// TIA Portal V20 export
FUNCTION_BLOCK "Sequence_4_STKInterface"   // FB181, LAD
TITLE = Sequence
// Sequence template programmend in ladder logic
// stored: IsIECCheckEnabled true, MemoryReserve 100, Namespace Unit1.Em7, SetENOAutomatically true
   VAR_OUTPUT
      safeState : Bool;
   END_VAR
   VAR_IN_OUT
      controlNodeStep : "LER_typeStep";
      controlNodeJobs : "LAF_typeJobs";
      controlNodeSequence : "LAF_typeSequence";
      HmiInterfaceJobs : "LAF_typeJobsInterface";
      HmiInterfaceSequence : "LAF_typeSequenceInterface";
      PartDataStkPpPos : "LER_typePartData";
      InterfaceR2SData : "LER_typeCommunicationR2SData";
      InterfaceS2RData : "LER_typeCommunicationS2RData";
   END_VAR
   VAR
      instSequenceLADControl { ExternalWritable := 'False'} : "LAF_ControlLadSequence";
      instSequenceLADStatus { ExternalWritable := 'False'} : "LAF_StatusLadSequence";
      statPulse { ExternalWritable := 'False'} : Array[0..999] of Bool;
      statTonTimer { ExternalWritable := 'False'} : Array[0..999] of TON_TIME;
   END_VAR
   VAR_TEMP
      tempCustomerAction : Bool;   // Placeholder for possible actions
      tempDo_nothing_and_wait_for_init : Bool;   // Placeholder for doing nothing
      tempSafeStateCondition : Bool;   // Temp Condition for the equipment module to be in a safe state
      tempPartDataStkPpPos : "LER_typePartData";
   END_VAR
   VAR CONSTANT
      STEP_IDLE : DInt := 1;   // Idle Step
      JOB_1_STEP_01 : DInt := 101;
      JOB_1_STEP_11 : DInt := 111;
      JOB_1_STEP_21 : DInt := 121;
      JOB_1_STEP_31 : DInt := 131;
      JOB_1_STEP_41 : DInt := 141;
      JOB_1_STEP_51 : DInt := 151;
      JOB_1_STEP_61 : DInt := 161;
      JOB_1_STEP_71 : DInt := 171;
      JOB_1_STEP_81 : DInt := 181;
      JOB_1_STEP_91 : DInt := 191;
      JOB_2_STEP_01 : DInt := 201;
      JOB_2_STEP_11 : DInt := 211;
      JOB_2_STEP_21 : DInt := 221;
      JOB_2_STEP_31 : DInt := 231;
      JOB_2_STEP_41 : DInt := 241;
      JOB_2_STEP_51 : DInt := 251;
      JOB_2_STEP_61 : DInt := 261;
      JOB_2_STEP_71 : DInt := 271;
      JOB_2_STEP_81 : DInt := 281;
      JOB_2_STEP_91 : DInt := 291;
      JOB_3_STEP_01 : DInt := 301;
      JOB_3_STEP_11 : DInt := 311;
      JOB_3_STEP_21 : DInt := 321;
      JOB_3_STEP_31 : DInt := 331;
      JOB_3_STEP_41 : DInt := 341;
      JOB_3_STEP_51 : DInt := 351;
      JOB_3_STEP_61 : DInt := 361;
      JOB_3_STEP_71 : DInt := 371;
      JOB_3_STEP_81 : DInt := 381;
      JOB_3_STEP_91 : DInt := 391;
      JOB_4_STEP_01 : DInt := 401;
      JOB_4_STEP_11 : DInt := 411;
      JOB_4_STEP_21 : DInt := 421;
      JOB_4_STEP_31 : DInt := 431;
      JOB_4_STEP_41 : DInt := 441;
      JOB_4_STEP_51 : DInt := 451;
      JOB_4_STEP_61 : DInt := 461;
      JOB_4_STEP_71 : DInt := 471;
      JOB_4_STEP_81 : DInt := 481;
      JOB_4_STEP_91 : DInt := 491;
      STEP_IMMEDIATE_STOP : DInt := 901;   // Step executed when an immediate stop command is triggered for the sequence (i.e. when unit is in state aborting)
      SeqDelayTime : Time := T#100ms;
      SeqNoDelayTime : Time;
      TRUE : Bool := TRUE;
      FALSE : Bool := FALSE;
   END_VAR
   // // InterfaceR2SData.InterfaceData."Bool"[0] : Load Enable
   // // InterfaceR2SData.InterfaceData."Bool"[1] : Load Complete Comfirm
   // // InterfaceR2SData.InterfaceData."Bool"[2] : Cell Data Report
   // // InterfaceR2SData.InterfaceData."Bool"[10] : CollisionAreaOn
   // // InterfaceR2SData.InterfaceData."Bool"[11] : CollisionAreaOff
   // // InterfaceR2SData.InterfaceData."Bool"[15] : HeartBeat
   // // InterfaceS2RData.InterfaceData."Bool"[0] : Load Requset
   // // InterfaceS2RData.InterfaceData."Bool"[1] : Load Busy
   // // InterfaceS2RData.InterfaceData."Bool"[2] : Load Complete
   // // InterfaceS2RData.InterfaceData."Bool"[3] : Cell Data Request
   // // InterfaceS2RData.InterfaceData."Bool"[4] : Cell Data Report Ack
   // // InterfaceS2RData.InterfaceData."Bool"[5] : Cell Data Report Nck
   VAR_TEMP   // added for the SCL form of the ladder/FBD networks
      _w1 : Bool;
      _w2 : Bool;
      _w3 : Bool;
   END_VAR
BEGIN

REGION Network 1: BLOCK INFO HEADER
   // (company) / (C) Copyright (year)
   // ---------------------------------------------------------------------------------
   // Title:                             (Title of this block)
   // Comment/Function: (that is implemented in the block)
   // Library/Family:           (that the source is dedicated to)
   // Author:                        (department / person in charge / contact)
   // Target System:          (test system with FW version)
   // Engineering:              TIA Portal (SW version)
   // Restrictions:               (OB types, etc.)
   // Requirements:           (hardware, technological package, etc.)
   // ---------------------------------------------------------------------------------
   // Change log table:
   // Version          | Date             | Signature      | Expert in charge  | Changes applied ------------------------|----------------------|-------------------------|--------------------------------|-----------------------
   // 001.000.000 | yyyy-mm-dd | 0x00000000 | (name of expert) | First released version
END_REGION

REGION Network 2: DESCRIPTION
   // This is a template block provided by the Automation Framework. It can be used to create an own project.
   // The Block Info Header is prepared to put in your own data.
   // Description of the block could be added here and the docu created by Code2Docu.
END_REGION

REGION Network 3: *************** CONTROL **********************
END_REGION

REGION Network 4: Sequence Control
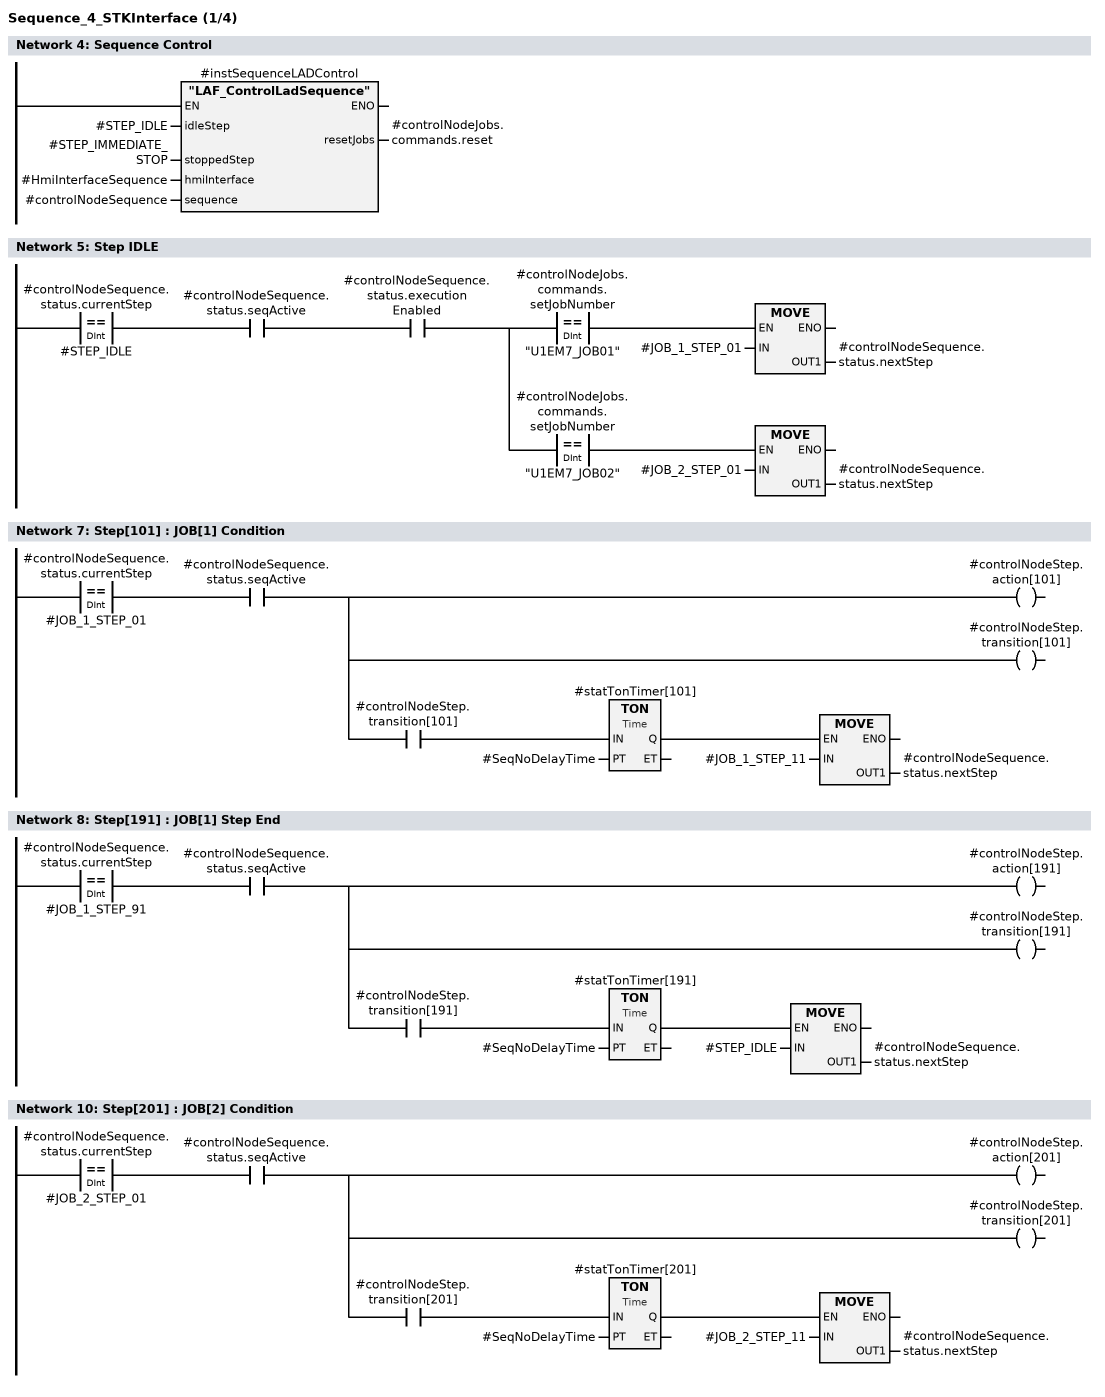
   RUNG wire#powerrail
      #instSequenceLADControl(idleStep := #STEP_IDLE, stoppedStep := #STEP_IMMEDIATE_STOP, hmiInterface := #HmiInterfaceSequence, sequence := #controlNodeSequence, resetJobs => #controlNodeJobs.commands.reset)
   END_RUNG
   // the same network as SCL:
   #instSequenceLADControl(idleStep := #STEP_IDLE,   // "LAF_ControlLadSequence"
                           stoppedStep := #STEP_IMMEDIATE_STOP,
                           hmiInterface := #HmiInterfaceSequence,
                           sequence := #controlNodeSequence,
                           resetJobs => #controlNodeJobs.commands.reset);
END_REGION

REGION Network 5: Step IDLE
   RUNG wire#powerrail
      { S7_Templates := "SrcType := DInt" } EQ_Contact(in1 := #controlNodeSequence.status.currentStep, in2 := #STEP_IDLE)
      Contact( #controlNodeSequence.status.seqActive )
      Contact( #controlNodeSequence.status.executionEnabled )
      wire#w1
      { S7_Templates := "SrcType := DInt" } EQ_Contact(in1 := #controlNodeJobs.commands.setJobNumber, in2 := "U1EM7_JOB01")
      Move(in := #JOB_1_STEP_01, out1 => #controlNodeSequence.status.nextStep)
   END_RUNG
   RUNG wire#w1
      { S7_Templates := "SrcType := DInt" } EQ_Contact(in1 := #controlNodeJobs.commands.setJobNumber, in2 := "U1EM7_JOB02")
      Move(in := #JOB_2_STEP_01, out1 => #controlNodeSequence.status.nextStep)
   END_RUNG
   // the same network as SCL:
   #_w1 := (#controlNodeSequence.status.currentStep = #STEP_IDLE) AND #controlNodeSequence.status.seqActive AND #controlNodeSequence.status.executionEnabled;
   IF #_w1 AND (#controlNodeJobs.commands.setJobNumber = "U1EM7_JOB01") THEN
       #controlNodeSequence.status.nextStep := #JOB_1_STEP_01;
   END_IF;
   IF #_w1 AND (#controlNodeJobs.commands.setJobNumber = "U1EM7_JOB02") THEN
       #controlNodeSequence.status.nextStep := #JOB_2_STEP_01;
   END_IF;
END_REGION

REGION Network 6: ******************** JOB[1] EM INITIALIZED ********************
END_REGION

REGION Network 7: Step[101] : JOB[1] Condition
   RUNG wire#powerrail
      { S7_Templates := "SrcType := DInt" } EQ_Contact(in1 := #controlNodeSequence.status.currentStep, in2 := #JOB_1_STEP_01)
      Contact( #controlNodeSequence.status.seqActive )
      wire#w1
      Coil( #controlNodeStep.action[101] )
   END_RUNG
   RUNG wire#w1
      Coil( #controlNodeStep.transition[101] )
   END_RUNG
   RUNG wire#w1
      Contact( #controlNodeStep.transition[101] )
      { S7_Templates := "time_type := Time" } #statTonTimer[101].TON(pt := #SeqNoDelayTime, et =>)
      Move(in := #JOB_1_STEP_11, out1 => #controlNodeSequence.status.nextStep)
   END_RUNG
   // the same network as SCL:
   #controlNodeStep.action[101] := (#controlNodeSequence.status.currentStep = #JOB_1_STEP_01) AND #controlNodeSequence.status.seqActive;
   #controlNodeStep.transition[101] := (#controlNodeSequence.status.currentStep = #JOB_1_STEP_01) AND #controlNodeSequence.status.seqActive;
   #statTonTimer[101].TON(IN := (#controlNodeSequence.status.currentStep = #JOB_1_STEP_01) AND #controlNodeSequence.status.seqActive AND #controlNodeStep.transition[101],
                          PT := #SeqNoDelayTime);
   IF #statTonTimer[101].Q THEN #controlNodeSequence.status.nextStep := #JOB_1_STEP_11; END_IF;
END_REGION

REGION Network 8: Step[191] : JOB[1] Step End
   RUNG wire#powerrail
      { S7_Templates := "SrcType := DInt" } EQ_Contact(in1 := #controlNodeSequence.status.currentStep, in2 := #JOB_1_STEP_91)
      Contact( #controlNodeSequence.status.seqActive )
      wire#w1
      Coil( #controlNodeStep.action[191] )
   END_RUNG
   RUNG wire#w1
      Coil( #controlNodeStep.transition[191] )
   END_RUNG
   RUNG wire#w1
      Contact( #controlNodeStep.transition[191] )
      { S7_Templates := "time_type := Time" } #statTonTimer[191].TON(pt := #SeqNoDelayTime, et =>)
      Move(in := #STEP_IDLE, out1 => #controlNodeSequence.status.nextStep)
   END_RUNG
   // the same network as SCL:
   #controlNodeStep.action[191] := (#controlNodeSequence.status.currentStep = #JOB_1_STEP_91) AND #controlNodeSequence.status.seqActive;
   #controlNodeStep.transition[191] := (#controlNodeSequence.status.currentStep = #JOB_1_STEP_91) AND #controlNodeSequence.status.seqActive;
   #statTonTimer[191].TON(IN := (#controlNodeSequence.status.currentStep = #JOB_1_STEP_91) AND #controlNodeSequence.status.seqActive AND #controlNodeStep.transition[191],
                          PT := #SeqNoDelayTime);
   IF #statTonTimer[191].Q THEN #controlNodeSequence.status.nextStep := #STEP_IDLE; END_IF;
END_REGION

REGION Network 9: ******************** JOB[2] STACK INTERFACE AUTO ********************
END_REGION

REGION Network 10: Step[201] : JOB[2] Condition
   RUNG wire#powerrail
      { S7_Templates := "SrcType := DInt" } EQ_Contact(in1 := #controlNodeSequence.status.currentStep, in2 := #JOB_2_STEP_01)
      Contact( #controlNodeSequence.status.seqActive )
      wire#w1
      Coil( #controlNodeStep.action[201] )
   END_RUNG
   RUNG wire#w1
      Coil( #controlNodeStep.transition[201] )
   END_RUNG
   RUNG wire#w1
      Contact( #controlNodeStep.transition[201] )
      { S7_Templates := "time_type := Time" } #statTonTimer[201].TON(pt := #SeqNoDelayTime, et =>)
      Move(in := #JOB_2_STEP_11, out1 => #controlNodeSequence.status.nextStep)
   END_RUNG
   // the same network as SCL:
   #controlNodeStep.action[201] := (#controlNodeSequence.status.currentStep = #JOB_2_STEP_01) AND #controlNodeSequence.status.seqActive;
   #controlNodeStep.transition[201] := (#controlNodeSequence.status.currentStep = #JOB_2_STEP_01) AND #controlNodeSequence.status.seqActive;
   #statTonTimer[201].TON(IN := (#controlNodeSequence.status.currentStep = #JOB_2_STEP_01) AND #controlNodeSequence.status.seqActive AND #controlNodeStep.transition[201],
                          PT := #SeqNoDelayTime);
   IF #statTonTimer[201].Q THEN #controlNodeSequence.status.nextStep := #JOB_2_STEP_11; END_IF;
END_REGION

REGION Network 11: Step[211] : Load Requset
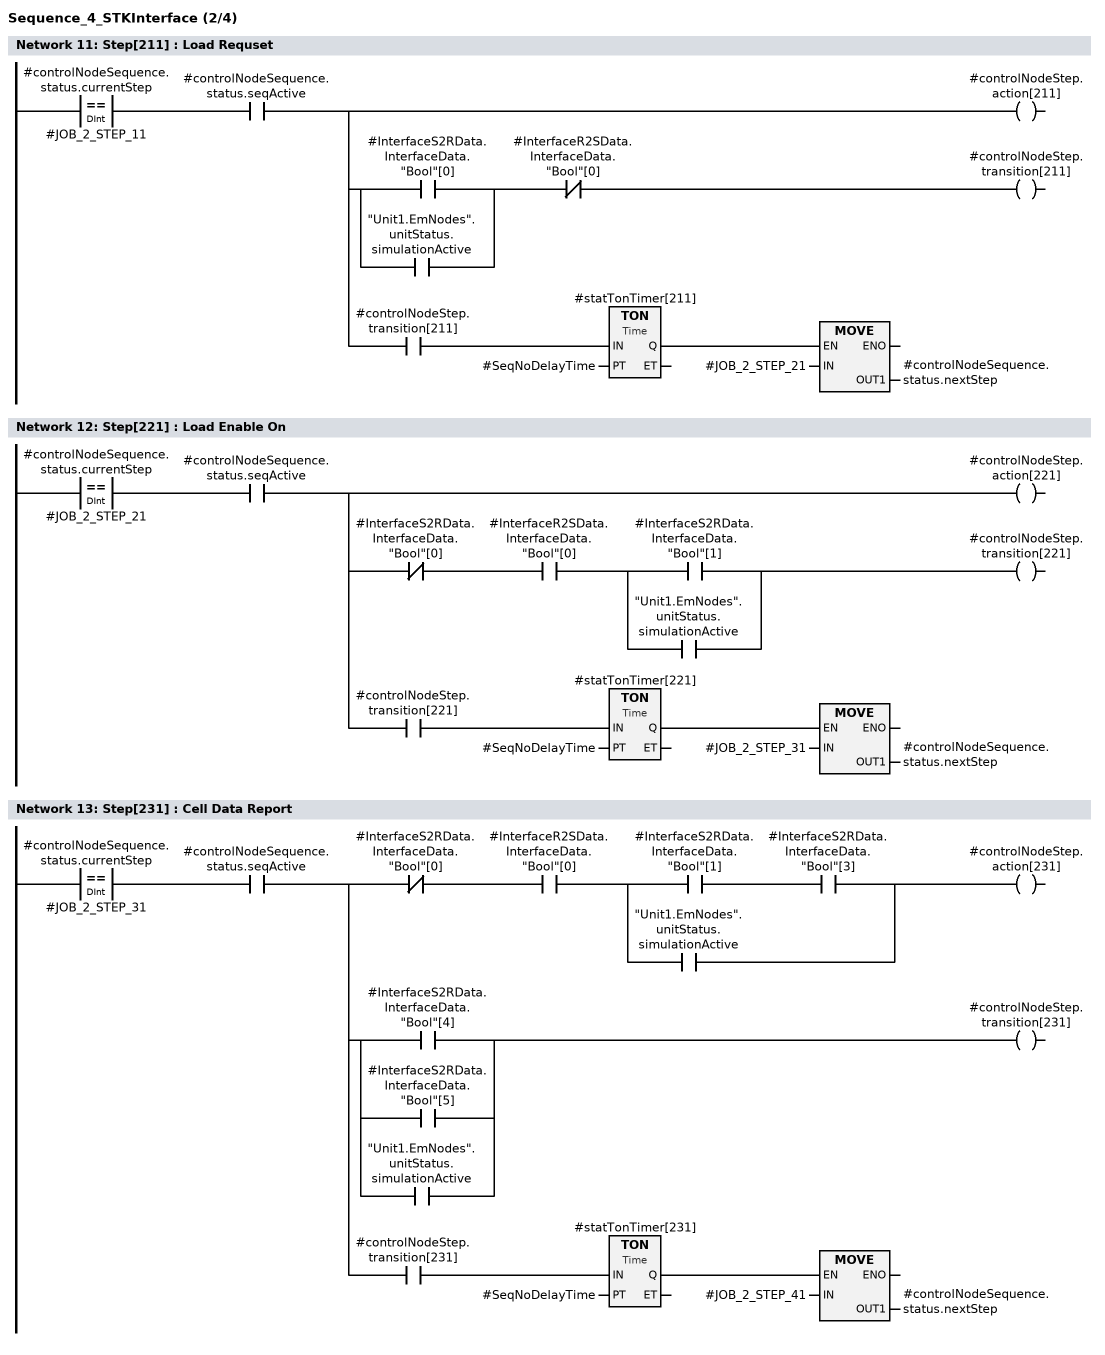
   RUNG wire#powerrail
      { S7_Templates := "SrcType := DInt" } EQ_Contact(in1 := #controlNodeSequence.status.currentStep, in2 := #JOB_2_STEP_11)
      Contact( #controlNodeSequence.status.seqActive )
      wire#w1
      Coil( #controlNodeStep.action[211] )
   END_RUNG
   RUNG wire#w1
      Contact( #InterfaceS2RData.InterfaceData."Bool"[0] )
      wire#w2
      I_Contact( #InterfaceR2SData.InterfaceData."Bool"[0] )
      Coil( #controlNodeStep.transition[211] )
   END_RUNG
   RUNG wire#w1
      Contact( "Unit1.EmNodes".unitStatus.simulationActive )
   END_RUNG wire#w2
   RUNG wire#w1
      Contact( #controlNodeStep.transition[211] )
      { S7_Templates := "time_type := Time" } #statTonTimer[211].TON(pt := #SeqNoDelayTime, et =>)
      Move(in := #JOB_2_STEP_21, out1 => #controlNodeSequence.status.nextStep)
   END_RUNG
   // the same network as SCL:
   #controlNodeStep.action[211] := (#controlNodeSequence.status.currentStep = #JOB_2_STEP_11) AND #controlNodeSequence.status.seqActive;
   #controlNodeStep.transition[211] := (#controlNodeSequence.status.currentStep = #JOB_2_STEP_11) AND #controlNodeSequence.status.seqActive AND (#InterfaceS2RData.InterfaceData."Bool"[0] OR "Unit1.EmNodes".unitStatus.simulationActive) AND NOT #InterfaceR2SData.InterfaceData."Bool"[0];
   #statTonTimer[211].TON(IN := (#controlNodeSequence.status.currentStep = #JOB_2_STEP_11) AND #controlNodeSequence.status.seqActive AND #controlNodeStep.transition[211],
                          PT := #SeqNoDelayTime);
   IF #statTonTimer[211].Q THEN #controlNodeSequence.status.nextStep := #JOB_2_STEP_21; END_IF;
END_REGION

REGION Network 12: Step[221] : Load Enable On
   RUNG wire#powerrail
      { S7_Templates := "SrcType := DInt" } EQ_Contact(in1 := #controlNodeSequence.status.currentStep, in2 := #JOB_2_STEP_21)
      Contact( #controlNodeSequence.status.seqActive )
      wire#w1
      Coil( #controlNodeStep.action[221] )
   END_RUNG
   RUNG wire#w1
      I_Contact( #InterfaceS2RData.InterfaceData."Bool"[0] )
      Contact( #InterfaceR2SData.InterfaceData."Bool"[0] )
      wire#w2
      Contact( #InterfaceS2RData.InterfaceData."Bool"[1] )
      wire#w3
      Coil( #controlNodeStep.transition[221] )
   END_RUNG
   RUNG wire#w2
      Contact( "Unit1.EmNodes".unitStatus.simulationActive )
   END_RUNG wire#w3
   RUNG wire#w1
      Contact( #controlNodeStep.transition[221] )
      { S7_Templates := "time_type := Time" } #statTonTimer[221].TON(pt := #SeqNoDelayTime, et =>)
      Move(in := #JOB_2_STEP_31, out1 => #controlNodeSequence.status.nextStep)
   END_RUNG
   // the same network as SCL:
   #controlNodeStep.action[221] := (#controlNodeSequence.status.currentStep = #JOB_2_STEP_21) AND #controlNodeSequence.status.seqActive;
   #controlNodeStep.transition[221] := (#controlNodeSequence.status.currentStep = #JOB_2_STEP_21) AND #controlNodeSequence.status.seqActive AND NOT #InterfaceS2RData.InterfaceData."Bool"[0] AND #InterfaceR2SData.InterfaceData."Bool"[0] AND (#InterfaceS2RData.InterfaceData."Bool"[1] OR "Unit1.EmNodes".unitStatus.simulationActive);
   #statTonTimer[221].TON(IN := (#controlNodeSequence.status.currentStep = #JOB_2_STEP_21) AND #controlNodeSequence.status.seqActive AND #controlNodeStep.transition[221],
                          PT := #SeqNoDelayTime);
   IF #statTonTimer[221].Q THEN #controlNodeSequence.status.nextStep := #JOB_2_STEP_31; END_IF;
END_REGION

REGION Network 13: Step[231] : Cell Data Report
   RUNG wire#powerrail
      { S7_Templates := "SrcType := DInt" } EQ_Contact(in1 := #controlNodeSequence.status.currentStep, in2 := #JOB_2_STEP_31)
      Contact( #controlNodeSequence.status.seqActive )
      wire#w1
      I_Contact( #InterfaceS2RData.InterfaceData."Bool"[0] )
      Contact( #InterfaceR2SData.InterfaceData."Bool"[0] )
      wire#w2
      Contact( #InterfaceS2RData.InterfaceData."Bool"[1] )
      Contact( #InterfaceS2RData.InterfaceData."Bool"[3] )
      wire#w3
      Coil( #controlNodeStep.action[231] )
   END_RUNG
   RUNG wire#w2
      Contact( "Unit1.EmNodes".unitStatus.simulationActive )
   END_RUNG wire#w3
   RUNG wire#w1
      Contact( #InterfaceS2RData.InterfaceData."Bool"[4] )
      wire#w4
      Coil( #controlNodeStep.transition[231] )
   END_RUNG
   RUNG wire#w1
      Contact( #InterfaceS2RData.InterfaceData."Bool"[5] )
   END_RUNG wire#w4
   RUNG wire#w1
      Contact( "Unit1.EmNodes".unitStatus.simulationActive )
   END_RUNG wire#w4
   RUNG wire#w1
      Contact( #controlNodeStep.transition[231] )
      { S7_Templates := "time_type := Time" } #statTonTimer[231].TON(pt := #SeqNoDelayTime, et =>)
      Move(in := #JOB_2_STEP_41, out1 => #controlNodeSequence.status.nextStep)
   END_RUNG
   // the same network as SCL:
   #_w1 := (#controlNodeSequence.status.currentStep = #JOB_2_STEP_31) AND #controlNodeSequence.status.seqActive;
   #controlNodeStep.action[231] := #_w1 AND NOT #InterfaceS2RData.InterfaceData."Bool"[0] AND #InterfaceR2SData.InterfaceData."Bool"[0] AND ((#InterfaceS2RData.InterfaceData."Bool"[1] AND #InterfaceS2RData.InterfaceData."Bool"[3]) OR "Unit1.EmNodes".unitStatus.simulationActive);
   #controlNodeStep.transition[231] := #_w1 AND (#InterfaceS2RData.InterfaceData."Bool"[4] OR #InterfaceS2RData.InterfaceData."Bool"[5] OR "Unit1.EmNodes".unitStatus.simulationActive);
   #statTonTimer[231].TON(IN := #_w1 AND #controlNodeStep.transition[231], PT := #SeqNoDelayTime);
   IF #statTonTimer[231].Q THEN #controlNodeSequence.status.nextStep := #JOB_2_STEP_41; END_IF;
END_REGION

REGION Network 14: Step[241] : Load Enable Off
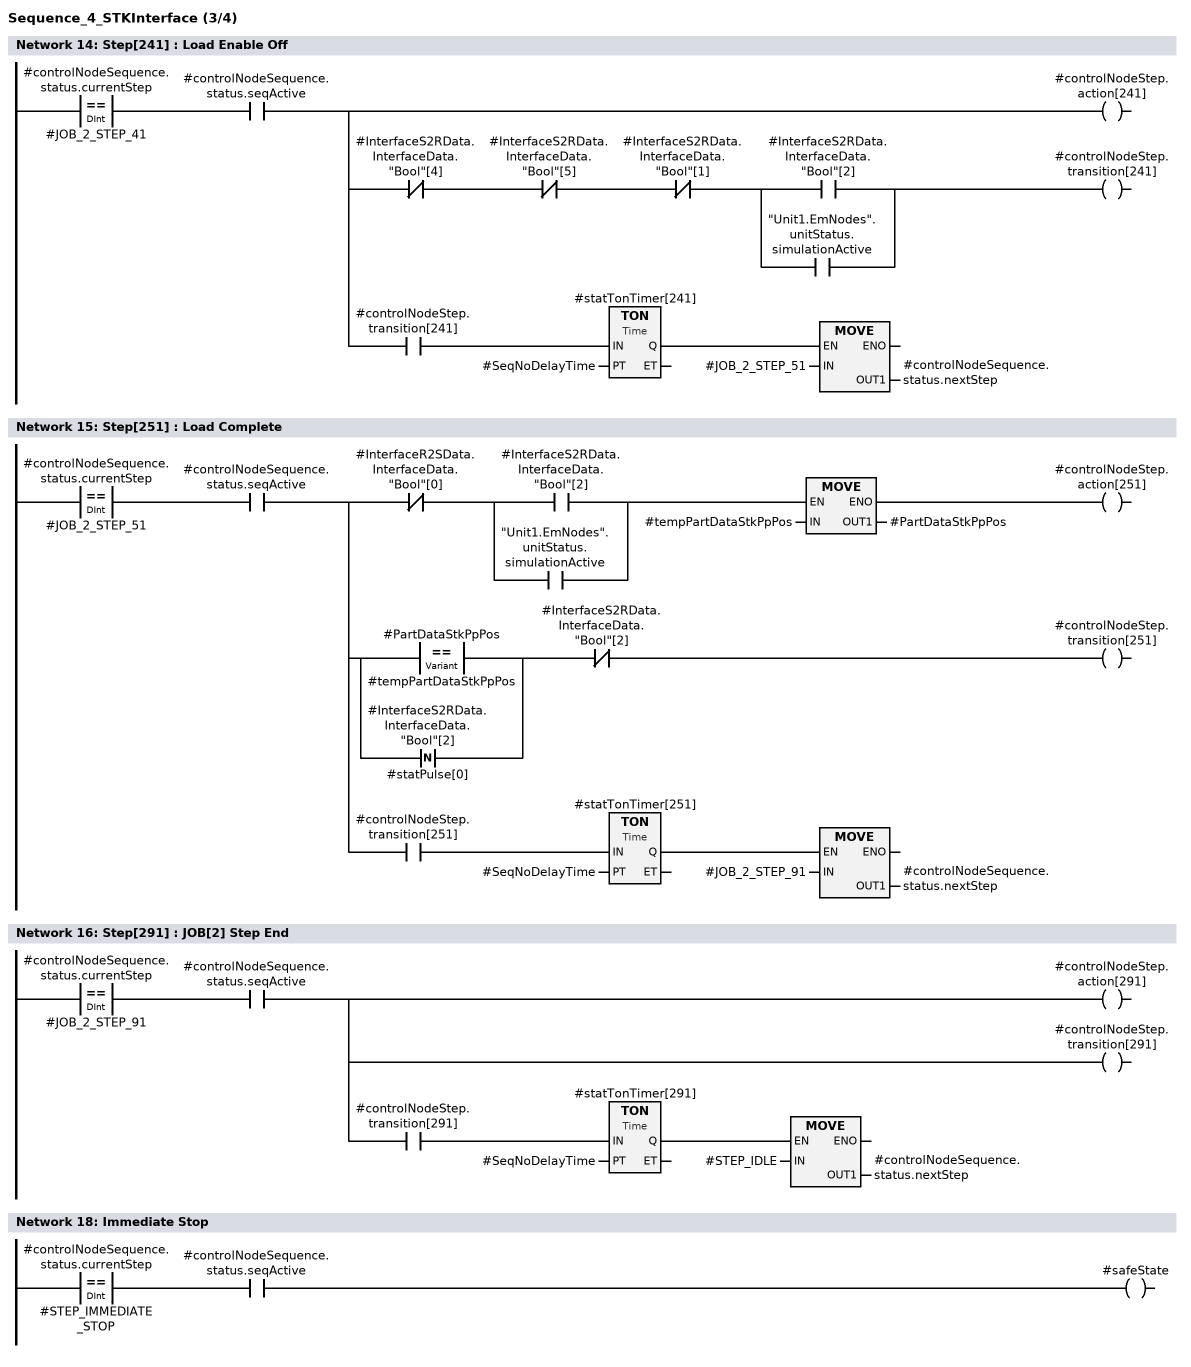
   RUNG wire#powerrail
      { S7_Templates := "SrcType := DInt" } EQ_Contact(in1 := #controlNodeSequence.status.currentStep, in2 := #JOB_2_STEP_41)
      Contact( #controlNodeSequence.status.seqActive )
      wire#w1
      Coil( #controlNodeStep.action[241] )
   END_RUNG
   RUNG wire#w1
      I_Contact( #InterfaceS2RData.InterfaceData."Bool"[4] )
      I_Contact( #InterfaceS2RData.InterfaceData."Bool"[5] )
      I_Contact( #InterfaceS2RData.InterfaceData."Bool"[1] )
      wire#w2
      Contact( #InterfaceS2RData.InterfaceData."Bool"[2] )
      wire#w3
      Coil( #controlNodeStep.transition[241] )
   END_RUNG
   RUNG wire#w2
      Contact( "Unit1.EmNodes".unitStatus.simulationActive )
   END_RUNG wire#w3
   RUNG wire#w1
      Contact( #controlNodeStep.transition[241] )
      { S7_Templates := "time_type := Time" } #statTonTimer[241].TON(pt := #SeqNoDelayTime, et =>)
      Move(in := #JOB_2_STEP_51, out1 => #controlNodeSequence.status.nextStep)
   END_RUNG
   // the same network as SCL:
   #controlNodeStep.action[241] := (#controlNodeSequence.status.currentStep = #JOB_2_STEP_41) AND #controlNodeSequence.status.seqActive;
   #controlNodeStep.transition[241] := (#controlNodeSequence.status.currentStep = #JOB_2_STEP_41) AND #controlNodeSequence.status.seqActive AND NOT #InterfaceS2RData.InterfaceData."Bool"[4] AND NOT #InterfaceS2RData.InterfaceData."Bool"[5] AND NOT #InterfaceS2RData.InterfaceData."Bool"[1] AND (#InterfaceS2RData.InterfaceData."Bool"[2] OR "Unit1.EmNodes".unitStatus.simulationActive);
   #statTonTimer[241].TON(IN := (#controlNodeSequence.status.currentStep = #JOB_2_STEP_41) AND #controlNodeSequence.status.seqActive AND #controlNodeStep.transition[241],
                          PT := #SeqNoDelayTime);
   IF #statTonTimer[241].Q THEN #controlNodeSequence.status.nextStep := #JOB_2_STEP_51; END_IF;
END_REGION

REGION Network 15: Step[251] : Load Complete
   RUNG wire#powerrail
      { S7_Templates := "SrcType := DInt" } EQ_Contact(in1 := #controlNodeSequence.status.currentStep, in2 := #JOB_2_STEP_51)
      Contact( #controlNodeSequence.status.seqActive )
      wire#w1
      I_Contact( #InterfaceR2SData.InterfaceData."Bool"[0] )
      wire#w2
      Contact( #InterfaceS2RData.InterfaceData."Bool"[2] )
      wire#w3
      Move(in := #tempPartDataStkPpPos, out1 => #PartDataStkPpPos)
      Coil( #controlNodeStep.action[251] )
   END_RUNG
   RUNG wire#w2
      Contact( "Unit1.EmNodes".unitStatus.simulationActive )
   END_RUNG wire#w3
   RUNG wire#w1
      { S7_Templates := "SrcType := Variant" } EQ_Contact(in1 := #PartDataStkPpPos, in2 := #tempPartDataStkPpPos)
      wire#w4
      I_Contact( #InterfaceS2RData.InterfaceData."Bool"[2] )
      Coil( #controlNodeStep.transition[251] )
   END_RUNG
   RUNG wire#w1
      N_Contact(operand := #InterfaceS2RData.InterfaceData."Bool"[2], bit := #statPulse[0])
   END_RUNG wire#w4
   RUNG wire#w1
      Contact( #controlNodeStep.transition[251] )
      { S7_Templates := "time_type := Time" } #statTonTimer[251].TON(pt := #SeqNoDelayTime, et =>)
      Move(in := #JOB_2_STEP_91, out1 => #controlNodeSequence.status.nextStep)
   END_RUNG
   // the same network as SCL:
   #_w1 := (#controlNodeSequence.status.currentStep = #JOB_2_STEP_51) AND #controlNodeSequence.status.seqActive;
   #_w2 := #_w1 AND NOT #InterfaceR2SData.InterfaceData."Bool"[0] AND (#InterfaceS2RData.InterfaceData."Bool"[2] OR "Unit1.EmNodes".unitStatus.simulationActive);
   IF #_w2 THEN #PartDataStkPpPos := #tempPartDataStkPpPos; END_IF;
   #controlNodeStep.action[251] := #_w2;
   #_w3 := #_w1 AND NOT #InterfaceS2RData.InterfaceData."Bool"[2] AND #statPulse[0];   // falling edge of #InterfaceS2RData.InterfaceData."Bool"[2]
   #statPulse[0] := #InterfaceS2RData.InterfaceData."Bool"[2];
   #controlNodeStep.transition[251] := ((#_w1 AND (#PartDataStkPpPos = #tempPartDataStkPpPos)) OR #_w3) AND NOT #InterfaceS2RData.InterfaceData."Bool"[2];
   #statTonTimer[251].TON(IN := #_w1 AND #controlNodeStep.transition[251], PT := #SeqNoDelayTime);
   IF #statTonTimer[251].Q THEN #controlNodeSequence.status.nextStep := #JOB_2_STEP_91; END_IF;
END_REGION

REGION Network 16: Step[291] : JOB[2] Step End
   RUNG wire#powerrail
      { S7_Templates := "SrcType := DInt" } EQ_Contact(in1 := #controlNodeSequence.status.currentStep, in2 := #JOB_2_STEP_91)
      Contact( #controlNodeSequence.status.seqActive )
      wire#w1
      Coil( #controlNodeStep.action[291] )
   END_RUNG
   RUNG wire#w1
      Coil( #controlNodeStep.transition[291] )
   END_RUNG
   RUNG wire#w1
      Contact( #controlNodeStep.transition[291] )
      { S7_Templates := "time_type := Time" } #statTonTimer[291].TON(pt := #SeqNoDelayTime, et =>)
      Move(in := #STEP_IDLE, out1 => #controlNodeSequence.status.nextStep)
   END_RUNG
   // the same network as SCL:
   #controlNodeStep.action[291] := (#controlNodeSequence.status.currentStep = #JOB_2_STEP_91) AND #controlNodeSequence.status.seqActive;
   #controlNodeStep.transition[291] := (#controlNodeSequence.status.currentStep = #JOB_2_STEP_91) AND #controlNodeSequence.status.seqActive;
   #statTonTimer[291].TON(IN := (#controlNodeSequence.status.currentStep = #JOB_2_STEP_91) AND #controlNodeSequence.status.seqActive AND #controlNodeStep.transition[291],
                          PT := #SeqNoDelayTime);
   IF #statTonTimer[291].Q THEN #controlNodeSequence.status.nextStep := #STEP_IDLE; END_IF;
END_REGION

REGION Network 17: *************** IMMEDIATE STOP ****************
END_REGION

REGION Network 18: Immediate Stop
   RUNG wire#powerrail
      { S7_Templates := "SrcType := DInt" } EQ_Contact(in1 := #controlNodeSequence.status.currentStep, in2 := #STEP_IMMEDIATE_STOP)
      Contact( #controlNodeSequence.status.seqActive )
      Coil( #safeState )
   END_RUNG
   // the same network as SCL:
   #safeState := (#controlNodeSequence.status.currentStep = #STEP_IMMEDIATE_STOP) AND #controlNodeSequence.status.seqActive;
END_REGION

REGION Network 19: *************** STATUS **********************
END_REGION

REGION Network 20: Sequence Status
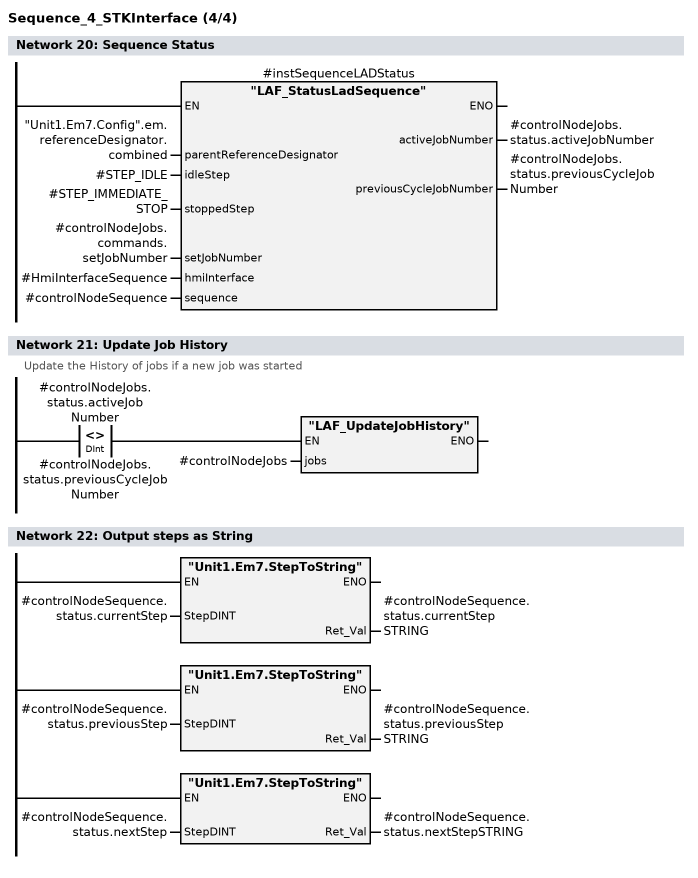
   RUNG wire#powerrail
      #instSequenceLADStatus(parentReferenceDesignator := "Unit1.Em7.Config".em.referenceDesignator.combined, idleStep := #STEP_IDLE, stoppedStep := #STEP_IMMEDIATE_STOP, setJobNumber := #controlNodeJobs.commands.setJobNumber, hmiInterface := #HmiInterfaceSequence, sequence := #controlNodeSequence, activeJobNumber => #controlNodeJobs.status.activeJobNumber, previousCycleJobNumber => #controlNodeJobs.status.previousCycleJobNumber)
   END_RUNG
   // the same network as SCL:
   #instSequenceLADStatus(parentReferenceDesignator := "Unit1.Em7.Config".em.referenceDesignator.combined,   // "LAF_StatusLadSequence"
                          idleStep := #STEP_IDLE,
                          stoppedStep := #STEP_IMMEDIATE_STOP,
                          setJobNumber := #controlNodeJobs.commands.setJobNumber,
                          hmiInterface := #HmiInterfaceSequence,
                          sequence := #controlNodeSequence,
                          activeJobNumber => #controlNodeJobs.status.activeJobNumber,
                          previousCycleJobNumber => #controlNodeJobs.status.previousCycleJobNumber);
END_REGION

REGION Network 21: Update Job History
   // Update the History of jobs if a new job was started
   RUNG wire#powerrail
      { S7_Templates := "SrcType := DInt" } NE_Contact(in1 := #controlNodeJobs.status.activeJobNumber, in2 := #controlNodeJobs.status.previousCycleJobNumber)
      "LAF_UpdateJobHistory"(jobs := #controlNodeJobs)
   END_RUNG
   // the same network as SCL:
   IF #controlNodeJobs.status.activeJobNumber <> #controlNodeJobs.status.previousCycleJobNumber THEN
       "LAF_UpdateJobHistory"(jobs := #controlNodeJobs);
   END_IF;
END_REGION

REGION Network 22: Output steps as String
   RUNG wire#powerrail
      "Unit1.Em7.StepToString"(StepDINT := #controlNodeSequence.status.currentStep, Ret_Val => #controlNodeSequence.status.currentStepSTRING)
   END_RUNG
   RUNG wire#powerrail
      "Unit1.Em7.StepToString"(StepDINT := #controlNodeSequence.status.previousStep, Ret_Val => #controlNodeSequence.status.previousStepSTRING)
   END_RUNG
   RUNG wire#powerrail
      "Unit1.Em7.StepToString"(StepDINT := #controlNodeSequence.status.nextStep, Ret_Val => #controlNodeSequence.status.nextStepSTRING)
   END_RUNG
   // the same network as SCL:
   #controlNodeSequence.status.currentStepSTRING := "Unit1.Em7.StepToString"(StepDINT := #controlNodeSequence.status.currentStep);
   #controlNodeSequence.status.previousStepSTRING := "Unit1.Em7.StepToString"(StepDINT := #controlNodeSequence.status.previousStep);
   #controlNodeSequence.status.nextStepSTRING := "Unit1.Em7.StepToString"(StepDINT := #controlNodeSequence.status.nextStep);
END_REGION
END_FUNCTION_BLOCK
